FUNCTION F_UpdateEventTimestampWithSystemTime
VAR_INPUT
	stEvent : REFERENCE TO ST_Event;
END_VAR
VAR
	fbGetSystemTime : GETSYSTEMTIME; //Get system time
	stFileTIme : T_FILETIME; //Filetime structure
END_VAR

fbGetSystemTIme(
	timeLoDW => stFileTIme.dwLowDateTime, 
	timeHiDW => stFileTIme.dwHighDateTime);
	
stEvent.dtTimestamp := FILETIME_TO_DT(fileTime := stFileTime);

END_FUNCTION

(* stored: Version 1.1.0.1
   POU F_UpdateEventTimestampWithSystemTime: Id {d37c28c3-1f20-4d00-b15c-7e62b46e36a7}, SpecialFunc None *)
